// TwinCAT 3 PLC project MixedSequentialAndParallelTests
// Title: TcUnit sequentially running tests example projects
// Company: www.tcunit.org
// Author: Jakob Sagatowski
// ProjectVersion: 1.0.0.0
// ProgramVersion: 3.1.4022.7
// libraries:
//   Tc2_Standard, * (Beckhoff Automation GmbH)
//   Tc2_System, * (Beckhoff Automation GmbH)
//   Tc3_Module, * (Beckhoff Automation GmbH)
//   TcUnit, * (www.tcunit.org)
// project tree:
//   GVLs/ GVL.TcGVL
//   / PlcTask.TcTTO
//   POUs/ FB_StateMachineFunctionBlock.TcPOU, FB_TimedFunctionBlock.TcPOU
//   Test/ FB_StateMachineAndTimedFunctionBlock_Test.TcPOU, PRG_TEST.TcPOU
// real-time tasks:
//   TASK PlcTask: cycle T#10ms, priority 20, ADS port 350

CONFIGURATION MixedSequentialAndParallelTests
    RESOURCE PLC ON TwinCAT3
        TASK PlcTask(INTERVAL := T#10ms, PRIORITY := 20);
        PROGRAM PRG_TEST WITH PlcTask : PRG_TEST;
    END_RESOURCE
END_CONFIGURATION

// ---- GVLs/GVL.TcGVL
{attribute 'qualified_only'}
// These variables only exist to test the TcUnit framework. You can ignore them.
VAR_GLOBAL
    nTimedFunctionBlockTestShortTime : ULINT;
    nTimedFunctionBlockTestLongTime : ULINT;
    nStateMachineFunctionBlockTestVariant100 : ULINT;
    nStateMachineFunctionBlockTestVariant50 : ULINT;
    nStateMachineFunctionBlockTestVariant20 : ULINT;
END_VAR

// ---- Test/PRG_TEST.TcPOU
(*
    This example executes four tests in a sequence, and on top of this there is also one test
    that runs in parallel with the other four tests. The execution of tests in a sequence is
    achieved by calling the TEST_ORDERED() for the four tests, and TEST() for the test that
    runs in parallel with the other. The test-order of the sequential tests is defined by the
    order of which the tests are being called. The tests include tests for function blocks
    which need several cycles to complete, as the function blocks under tests use both state
    machines and times to complete and to reach their correct output state.
*)
PROGRAM PRG_TEST
VAR
    StateMachineAndTimedFunctionBlock_Test : FB_StateMachineAndTimedFunctionBlock_Test;
END_VAR

TcUnit.RUN();

END_PROGRAM

// ---- Test/FB_StateMachineAndTimedFunctionBlock_Test.TcPOU
FUNCTION_BLOCK FB_StateMachineAndTimedFunctionBlock_Test EXTENDS TcUnit.FB_TestSuite

(* The tests are run in the order that they are called. Asserts are not evaluated before the previous test has called TEST_FINISHED() *)
TestShortTime(); // This test will fail
TestLongTime();
TestVariant100();
TestVariant50(); // This test runs in pararallel with the other four tests (which run in sequence)
TestVariant20(); // This test will fail

METHOD PRIVATE TestLongTime
(* We need to declare the FB_TimedFunctionBlock_Test as an instance variable,
   as it needs to hold its values over several cycles *)
VAR_INST
    // Function block under test
    fbTimedFunctionBlock : FB_TimedFunctionBlock;
    fbTon : TON := (PT := T#10S); // The maximum time we will run the test
END_VAR
VAR CONSTANT
    EXPECTED_RESULT : INT := 100;
END_VAR
(* Make sure to only run test logic if it's time for this test to execute *)
IF TEST_ORDERED('TestLongTime') THEN
    GVL.nTimedFunctionBlockTestLongTime := GVL.nTimedFunctionBlockTestLongTime + 1; // Only for testing the framework. Ignore this.
    fbTon(IN := TRUE); // Maximum time we will run the test
    fbTimedFunctionBlock(bExecute := TRUE);
    (* Check if we get a timeout or if we get the result we want *)
    IF fbTon.Q OR fbTimedFunctionBlock.nValue = EXPECTED_RESULT THEN
        AssertEquals_INT(Expected := EXPECTED_RESULT,
                         Actual := fbTimedFunctionBlock.nValue,
                         Message := 'Value not correct');
        TEST_FINISHED();
	END_IF
END_IF
END_METHOD

METHOD PRIVATE TestShortTime
(* We need to declare the FB_TimedFunctionBlock_Test as an instance variable,
   as it needs to hold its values over several cycles *)
VAR_INST
    // Function block under test
    fbTimedFunctionBlock : FB_TimedFunctionBlock;
    fbTon : TON := (PT := T#2S); // The maximum time we will run the test
END_VAR
VAR CONSTANT
    EXPECTED_RESULT : INT := 100;
END_VAR
(* Make sure to only run test logic if it's time for this test to execute
   Note that this test will fail, as we will not run it long enough to get the correct result! *)
IF TEST_ORDERED('TestShortTime') THEN
    GVL.nTimedFunctionBlockTestShortTime := GVL.nTimedFunctionBlockTestShortTime + 1; // Only for testing the framework. Ignore this.
    fbTon(IN := TRUE); // Maximum time we will run the test
    fbTimedFunctionBlock(bExecute := TRUE);
    (* Check if we get a timeout or if we get the result we want *)
    IF fbTon.Q OR fbTimedFunctionBlock.nValue = EXPECTED_RESULT THEN
        AssertEquals_INT(Expected := EXPECTED_RESULT,
                         Actual := fbTimedFunctionBlock.nValue,
                         Message := 'Value not correct');
        TEST_FINISHED();
	END_IF
END_IF
END_METHOD

METHOD PRIVATE TestVariant100
(* We need to declare the FB_StateMachineFunctionBlock as an instance variable,
   as it needs to hold its values over several cycles *)
VAR_INST
    // Function block under test
    fbStateMachineFunctionBlock : FB_StateMachineFunctionBlock;
    fbTon : TON := (PT := T#5S); // The maximum time we will run the test
END_VAR
VAR CONSTANT
    EXPECTED_RESULT : INT := 100;
END_VAR
// Make sure to only run test logic if it's time for this test to execute
IF TEST_ORDERED('TestVariant100') THEN
    GVL.nStateMachineFunctionBlockTestVariant100 := GVL.nStateMachineFunctionBlockTestVariant100 + 1; // Only for testing the framework. Ignore this.
    fbTon(IN := TRUE); // Maximum time we will run the test
    fbStateMachineFunctionBlock(bStart := TRUE, nVariant := 100);
    (* Check if we get a timeout or if we get the result we want *)
    IF fbTon.Q OR fbStateMachineFunctionBlock.nValue = EXPECTED_RESULT THEN
        AssertEquals_INT(Expected := EXPECTED_RESULT,
                         Actual := fbStateMachineFunctionBlock.nValue,
                         Message := 'Value not correct');
        TEST_FINISHED();
	END_IF
END_IF
END_METHOD

METHOD PRIVATE TestVariant20
(* We need to declare the FB_StateMachineFunctionBlock as an instance variable,
   as it needs to hold its values over several cycles *)
VAR_INST
    // Function block under test
    fbStateMachineFunctionBlock : FB_StateMachineFunctionBlock;
    fbTon : TON := (PT := T#1MS); // The maximum time we will run the test
END_VAR
VAR CONSTANT
    EXPECTED_RESULT : INT := 100;
END_VAR
(* Make sure to only run test logic if it's time for this test to execute
   Note that this test will fail, as we will not run it long enough to get the correct result! *)
IF TEST_ORDERED('TestVariant20') THEN
    GVL.nStateMachineFunctionBlockTestVariant20 := GVL.nStateMachineFunctionBlockTestVariant20 + 1; // Only for testing the framework. Ignore this.
    fbTon(IN := TRUE); // Maximum time we will run the test
    fbStateMachineFunctionBlock(bStart := TRUE, nVariant := 20);
    (* Check if we get a timeout or if we get the result we want *)
    IF fbTon.Q OR fbStateMachineFunctionBlock.nValue = EXPECTED_RESULT THEN
        AssertEquals_INT(Expected := EXPECTED_RESULT,
                         Actual := fbStateMachineFunctionBlock.nValue,
                         Message := 'Value not correct');
        TEST_FINISHED();
	END_IF
END_IF
END_METHOD

METHOD PRIVATE TestVariant50
(* We need to declare the FB_StateMachineFunctionBlock as an instance variable,
   as it needs to hold its values over several cycles *)
VAR_INST
    // Function block under test
    fbStateMachineFunctionBlock : FB_StateMachineFunctionBlock;
    fbTon : TON := (PT := T#5S); // The maximum time we will run the test
END_VAR
VAR CONSTANT
    EXPECTED_RESULT : INT := 200;
END_VAR
TEST('TestVariant50');
GVL.nStateMachineFunctionBlockTestVariant50 := GVL.nStateMachineFunctionBlockTestVariant50 + 1; // Only for testing the framework. Ignore this.
fbTon(IN := TRUE); // Maximum time we will run the test
fbStateMachineFunctionBlock(bStart := TRUE, nVariant := 50);
(* Check if we get a timeout or if we get the result we want *)
IF fbTon.Q OR fbStateMachineFunctionBlock.nValue = EXPECTED_RESULT THEN
    AssertEquals_INT(Expected := EXPECTED_RESULT,
                     Actual := fbStateMachineFunctionBlock.nValue,
                     Message := 'Value not correct');
    TEST_FINISHED();
END_IF
END_METHOD

END_FUNCTION_BLOCK

// ---- POUs/FB_TimedFunctionBlock.TcPOU
(* This test will return the nValue 100 when this function block has been executed with a rising edge of bStart for at least 10 seconds *)
FUNCTION_BLOCK FB_TimedFunctionBlock
VAR_INPUT
    bExecute : BOOL;
END_VAR
VAR_OUTPUT
    nValue : INT;
END_VAR
VAR
    fbTimer : Tc2_Standard.TON := (PT := T#5S);
END_VAR

fbTimer(IN := bExecute); // Start timer on high trigger, reset timer on low

// Return value 100 if timer elapsed, otherwise return value 0
IF fbTimer.Q THEN
    nValue := 100;
ELSE
    nValue := 0;
END_IF

END_FUNCTION_BLOCK

// ---- POUs/FB_StateMachineFunctionBlock.TcPOU
(* This function block will return a value after a couple of cycle calls, and after setting bStart to TRUE.
   It will return the value 100 if nVariant is set to anything else than 50, and the value 200 if nVariant is set to 50 *)
FUNCTION_BLOCK FB_StateMachineFunctionBlock
VAR_INPUT
    bStart : BOOL;
    nVariant : INT;
END_VAR
VAR_OUTPUT
    nValue : INT;
END_VAR
VAR
    nState : INT;
    bTrigger : R_TRIG();
END_VAR

CASE nState OF
    0 : 
        bTrigger(CLK := bStart);
        IF bTrigger.Q THEN
            nState := 1;
		END_IF

    1 :
        nValue := 0; // Reset output value
        nState := 2;

    2 :
        IF nVariant = 50 THEN
            nState := 20;
        ELSE
            nState := 10;
		END_IF

    10 :
        nValue := 100;
        nState := 0;

    20 :
        nValue := 200;
        nState := 0;
END_CASE

END_FUNCTION_BLOCK
